FUNCTION_BLOCK FutureMCMoveRelativeCreator IMPLEMENTS I_TaskCreator
VAR_INPUT
END_VAR
VAR_OUTPUT
END_VAR
VAR
	_axis: REFERENCE TO AXIS_REF;
	_distance : MC_LREAL;
	_velocity : MC_LREAL;
	_acceleration: MC_LREAL;
	_deceleration: MC_LREAL;
	_jerk		: MC_LREAL;
	_option : ST_MoveOptions;
	_buffer_mode : MC_BufferMode ;
END_VAR

{warning 'add method implementation '}
METHOD create_future : I_Future
VAR_INPUT
	(* Specify future name*)
	future_name	: STRING;
END_VAR
VAR
	_p_future : POINTER TO FutureMCMoveRelative;
END_VAR
_p_future := __NEW(FutureMCMoveRelative);
_p_future^.future_name := future_name;
_p_future^.set_parameters(_axis, _distance, _velocity, _acceleration, _deceleration,_jerk ,_buffer_mode);
_p_future^.set_options( _option);
create_future := _p_future^;
END_METHOD

{warning 'add method implementation '}
METHOD destroy_future : I_Future
VAR_INPUT
	(* Specify future instance whtat you want to delete.*)
	future	: I_Future;
END_VAR
VAR
	_p_future : POINTER TO FutureMCMoveRelative;
END_VAR
IF __QUERYPOINTER(future, _p_future) THEN
	__DELETE(_p_future);
	IF _p_future = 0  THEN
		destroy_future := 0;
	END_IF
END_IF
END_METHOD

METHOD set_options : BOOL
VAR_INPUT
	option : ST_MoveOptions;
END_VAR
_option := option;
END_METHOD

METHOD set_parameters : BOOL
VAR_INPUT
	axis : REFERENCE TO AXIS_REF;
	distance : MC_LREAL;
	velocity : MC_LREAL;
	acceleration	: MC_LREAL;		// Set deceleration in case let moving axis halt.
	deceleration	: MC_LREAL;		// Set deceleration in case let moving axis halt.
	jerk			: MC_LREAL;		// Set jerk in case let moving axis halt.
	buffer_mode : MC_BufferMode;
END_VAR
_axis REF= axis;
_distance := distance;
_velocity := velocity;
_acceleration := acceleration;
_deceleration := deceleration;
_jerk := jerk;
_buffer_mode := buffer_mode;
END_METHOD

END_FUNCTION_BLOCK

(* stored: Version 1.1.0.1, ProductVersion 3.1.4026.17
   POU FutureMCMoveRelativeCreator: Id {d645c079-a4a6-4ee0-a81e-ead6131d7763}, SpecialFunc None
   Method create_future: Id {0a940ebe-841c-4322-b2c6-27b95a617183}
   Method destroy_future: Id {902a1d6e-d586-4236-8491-52e82d8711c1}
   Method set_options: Id {3cb4e318-f02d-4de9-8ea6-6e24c0d34928}
   Method set_parameters: Id {28ce2ff1-d3a4-4e94-ac24-9c320f325ea1} *)
